TYPE T_AnyString : __SYSTEM.AnyType; END_TYPE

(* stored: Version 1.1.0.1
   DUT T_AnyString: Id {93cbf64c-702b-4fb9-9b4b-111d6df3de1f} *)
